FUNCTION TryConvert_UDINT_TO_UINT : BOOL
VAR_INPUT
	in : UDINT;
	out : REFERENCE TO UINT;
END_VAR

IF in > DatatypeLimits.MAX_VALUE_OF_UDINT_WHICH_CAN_BE_HELD_IN_A_UINT THEN
	RETURN;
END_IF

out := UDINT_TO_UINT(in);
TryConvert_UDINT_TO_UINT := TRUE;

END_FUNCTION

(* stored: Version 1.1.0.1, ProductVersion 3.1.4024.12
   POU TryConvert_UDINT_TO_UINT: Id {c9035e72-b749-4204-b652-06c6e251f1eb}, SpecialFunc None *)
